Staubli VAL3: JointBlend.pgx

program JointBlend()
begin
end
